{attribute 'qualified_only'}
VAR_GLOBAL
	FinishedWithSprayZoneSD1 : BOOL;
	FinishedWithSprayZoneSD2 : BOOL;
	
END_VAR

(* stored: Version 1.1.0.1, ProductVersion 3.1.4024.12
   GVL GVL_Job: Id {a6b4cce6-e948-4ea9-8c4a-f59817c3abc6} *)
